ABB RobotStudio station: RAPID Project.rspag

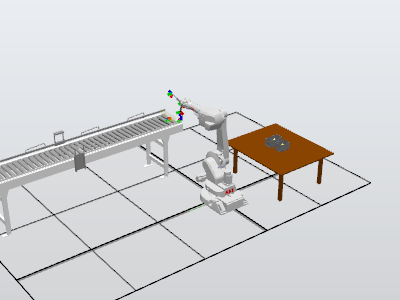
--- station ---
Station RAPID Project (saved by RobotStudio 23.4.10609.1)
Controller IRB1600_6_145
  mechanical unit ROB_1: IRB1600_6_145__03, 6 joints, base frame (0, 0, 0) mm
Layout (positions relative to the parent item):
  - IRB1600_6_145__03 [mechanism, from %ABB.RobotStudio.Models.IRB1600%\IRB1600_6_145_G_03.rslib] at (0, 0, 0) mm; joint values [0, 0, 0, 0, 0.5236, 0] (rad or m)
  - VacuumPenToolSC [smart component, from RAPID Project\VacuumPenToolSC.rslib] at (806.29, 0, 1154) mm, rotated rx 180 ry 60 rz 180 deg
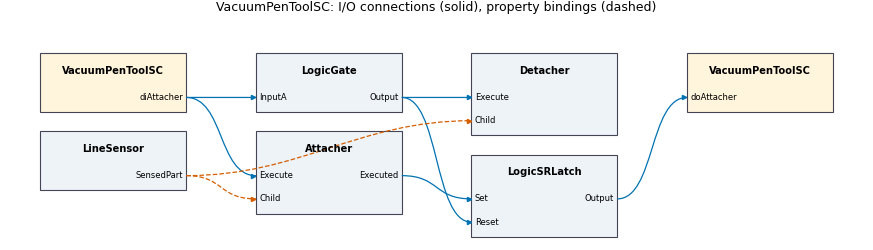
      connections:
        VacuumPenToolSC.diAttacher -> LogicGate.InputA
        LogicGate.Output -> Detacher.Execute
        Attacher.Executed -> LogicSRLatch.Set
        LogicSRLatch.Output -> VacuumPenToolSC.doAttacher
        VacuumPenToolSC.diAttacher -> Attacher.Execute
        LogicGate.Output -> LogicSRLatch.Reset
        LineSensor.SensedPart => Attacher.Child
        LineSensor.SensedPart => Detacher.Child
    - VacuumPenTool [mechanism, from RAPID Project\VacuumPenToolSC.rslib] at (0, 0, 0) mm
    - LineSensor [smart component, from Components\LineSensor.rslib]
        properties: Start=[0.107 -0.00037 0.127]; End=[0.114 0 0.134]; Radius=0.001; SensedPart=(none); SensedPoint=[0 0 0]; Length=0.00990640701768306; Tag=(none)
      - _sensorPart_ [part], size 8.4 x 2.4 x 8.4 mm
    - Attacher [smart component, from Components\Attacher.rslib]
        properties: Parent=VacuumPenTool; Flange=0; Child=(none); Mount=false; Offset=[0 0 0]; Orientation=[0 0 0]
    - Detacher [smart component, from Components\Detacher.rslib]
        properties: Child=(none); KeepPosition=true
    - LogicGate [smart component, from Components\LogicGate.rslib]
        properties: Operator=NOT; Delay=0
    - LogicSRLatch [smart component, from Components\LogicSRLatch.rslib]
  - mesa_marron [part] at (500, -500, 500) mm, rotated rx 90 ry 0 rz 180 deg, size 1200 x 500 x 1000 mm
  - box_big [part] at (1475.92, 2958.99, 0) mm, size 100 x 100 x 100 mm
  - box_small [part] at (1082.53, 3022.45, 0) mm, size 80 x 80 x 80 mm
  - Cardboard_container_bigSC [smart component]
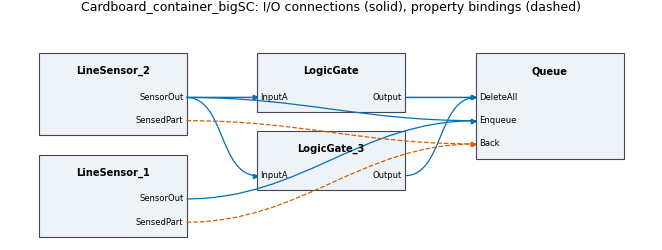
      connections:
        LineSensor_2.SensorOut -> LogicGate.InputA
        LogicGate.Output -> Queue.DeleteAll
        LineSensor_2.SensorOut -> LogicGate_2.InputA
        LogicGate_2.Output -> Queue.DeleteAll
        LineSensor_1.SensorOut -> Queue.Enqueue
        LineSensor_2.SensorOut -> Queue.Enqueue
        LineSensor_2.SensorOut -> LogicGate_3.InputA
        LogicGate_3.Output -> Queue.DeleteAll
        LineSensor_2.SensedPart => Queue.Back
        LineSensor_1.SensedPart => Queue.Back
    - UMS5_Cardboard_box_big_bottom [part] at (0, -1000, 521) mm, rotated rx 0 ry 0 rz -90 deg, size 220.2 x 110.8 x 110.2 mm
    - Queue [smart component, from Components\Queue.rslib]
        properties: Back=(none); Front=(none); Queue={6b8558fe-eb23-4042-ac4d-4b2e4693563e};{5ffcd9c3-88d3-497d-8378-cfc202dc5907};{29bb7ccf-0bc1-48a2-9f08-b9b634dbc6ca}; NumberOfObjects=1
    - LineSensor_1 [smart component, from Components\LineSensor.rslib]
        properties: Start=[0.05 -0.95 0.571]; End=[-0.05 -0.95 0.571]; Length=0.1; Radius=0; Tag=(none); SensedPart=(none); SensedPoint=[0.0499339485168457 -0.95 0.571]
      - _sensorPart_ [part], size 100 x 0 x 0 mm
    - LineSensor_2 [smart component, from Components\LineSensor.rslib]
        properties: Start=[0.05 -1.05 0.572]; End=[-0.05 -1.05 0.572]; Length=0.1; Radius=0; Tag=(none); SensedPart=(none); SensedPoint=[0 0 0]
      - _sensorPart_ [part], size 100 x 0 x 0 mm
    - LogicGate_3 [smart component, from Components\LogicGate.rslib]
        properties: Operator=NOP; Delay=4
  - Cardboard_container_smallSC [smart component]
      connections:
        LineSensor_3.SensorOut -> Queue_2.Enqueue
        LineSensor_4.SensorOut -> Queue_2.Enqueue
        LineSensor_4.SensorOut -> LogicGate_4.InputA
        LogicGate_4.Output -> Queue_2.DeleteAll
        LineSensor_3.SensedPart => Queue_2.Back
        LineSensor_4.SensedPart => Queue_2.Back
    - UMS5_Cardboard_box_small_bottom [part] at (-180, -1000, 521) mm, rotated rx 0 ry 0 rz -90 deg, size 180.2 x 110.8 x 110.2 mm
    - LineSensor_3 [smart component, from Components\LineSensor.rslib]
        properties: Start=[-0.23 -0.96 0.572]; End=[-0.13 -0.96 0.572]; Length=0.1; Radius=0; Tag=(none); SensedPart=(none); SensedPoint=[0 0 0]
      - _sensorPart_ [part], size 100 x 0 x 0 mm
    - LineSensor_4 [smart component, from Components\LineSensor.rslib]
        properties: Start=[-0.23 -1.04 0.572]; End=[-0.13 -1.04 0.572]; Length=0.1; Radius=0; Tag=(none); SensedPart=(none); SensedPoint=[0 0 0]
      - _sensorPart_ [part], size 100 x 0 x 0 mm
    - Queue_2 [smart component, from Components\Queue.rslib]
        properties: Back=(none); Front=(none); Queue=; NumberOfObjects=0
    - LogicGate_4 [smart component, from Components\LogicGate.rslib]
        properties: Operator=NOP; Delay=4
  - Conveyor [smart component] at (956.12, 2916.39, 0) mm, rotated rx 0 ry 0 rz -90 deg
      signals: DI start_or_resume, DO cube_ready, DO small_out, DO big_out
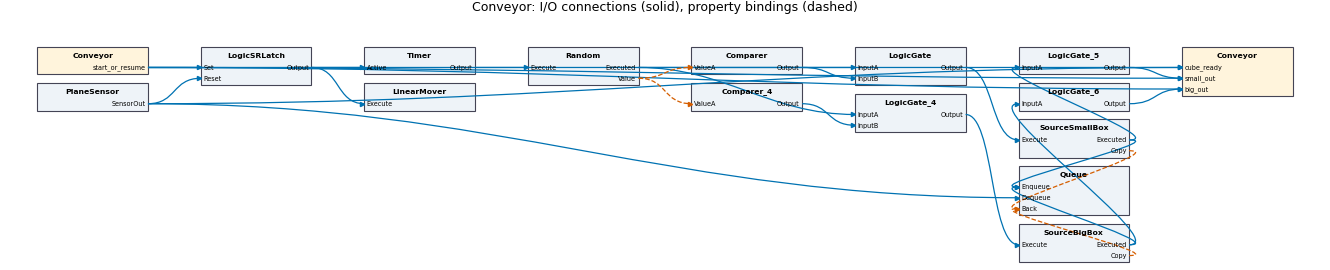
      connections:
        Timer.Output -> Random.Execute
        Random.Executed -> LogicGate.InputA
        Comparer.Output -> LogicGate.InputB
        Random.Executed -> LogicGate_4.InputA
        Comparer_4.Output -> LogicGate_4.InputB
        LogicGate.Output -> SourceSmallBox.Execute
        LogicGate_4.Output -> SourceBigBox.Execute
        SourceSmallBox.Executed -> Queue.Enqueue
        SourceBigBox.Executed -> Queue.Enqueue
        Conveyor.start_or_resume -> LogicSRLatch.Set
        PlaneSensor.SensorOut -> Queue.Dequeue
        PlaneSensor.SensorOut -> LogicSRLatch.Reset
        LogicSRLatch.Output -> Timer.Active
        LogicSRLatch.Output -> LinearMover.Execute
        PlaneSensor.SensorOut -> Conveyor.cube_ready
        SourceSmallBox.Executed -> LogicGate_5.InputA
        LogicGate_5.Output -> Conveyor.small_out
        SourceBigBox.Executed -> LogicGate_6.InputA
        LogicGate_6.Output -> Conveyor.big_out
        Conveyor.start_or_resume -> Conveyor.small_out
        Conveyor.start_or_resume -> Conveyor.big_out
        Conveyor.start_or_resume -> Conveyor.cube_ready
        Random.Value => Comparer.ValueA
        Random.Value => Comparer_4.ValueA
        SourceSmallBox.Copy => Queue.Back
        SourceBigBox.Copy => Queue.Back
    - SourceSmallBox [smart component, from Components\Source.rslib]
        properties: Source=box_small; Copy=(none); Parent=(none); Position=[1.118659 0.4 0.775]; Orientation=[0 0 0]; Transient=false; PhysicsBehavior=-1
    - SourceBigBox [smart component, from Components\Source.rslib]
        properties: Source=box_big; Copy=(none); Parent=(none); Position=[1.118659 0.4 0.775]; Orientation=[0 0 0]; Transient=false; PhysicsBehavior=-1
    - Random [smart component, from Components\Random.rslib]
        properties: Value=1.6316647863163; Min=0; Max=2
    - Comparer [smart component, from Components\Comparer.rslib]
        properties: ValueA=1.6316647863163; Operator=<=; ValueB=1
    - Timer [smart component, from Components\Timer.rslib]
        properties: StartTime=0; Interval=8; Repeat=true; CurrentTime=9.936
    - LogicGate [smart component, from Components\LogicGate.rslib]
        properties: Operator=AND; Delay=0
    - LogicGate_4 [smart component, from Components\LogicGate.rslib]
        properties: Operator=AND; Delay=0
    - Comparer_4 [smart component, from Components\Comparer.rslib]
        properties: ValueA=1.6316647863163; Operator=>; ValueB=1
    - Queue [smart component, from Components\Queue.rslib]
        properties: Back=(none); Front=(none); Queue={1131f909-5d82-4e84-bc9f-120231f9d299};{405f4df7-07e7-4b74-a1a1-a810a0d8cfa6};{743c33c0-6a87-4aec-9895-952089b91bbd};{216fa1ae-755b-4613-beaf-a983367b2fa7};{bf1b47c8-f294-4567-aa47-23f27967580f};{64bd0bdc-0a47-47ab-a397-a74a684aee1e};{437488d7-8282-475b-b486-389db32fdaa2};{671afbe1-b4fc-4869-acfd-eeadac196f1e};{a4dc94ab-7dff-4b2f-b405-15f84814c83e};{c4b58b1b-6de3-44d8-9367-5c715bdef502};{dda5cb65-1224-402a-bab3-4bfeb52fa140};{8990a0b7-37dc-4b49-b0cf-ca37f5f81eb5};{063f5e72-8178-40bf-9af7-13761aa78818};{318b9655-dbdc-41bc-a948-0739e52a5f4e};{94459ab9-d214-4441-90b7-aab42f321ec1};{846e7d94-1788-41a0-bce8-b7df51ff760f};{16d7a3a2-3dec-478f-b63b-07f1d7cc03de};{580626d5-5194-432f-9920-3f632f566f7d};{09cd6ac9-05a0-4cd8-820b-7021498e93a7};{8b0e4d5d-dbbf-4476-8b58-1e0bb391d2bd};{72ea86c5-dea0-4016-afa7-4ec3a2f95cb2};{db5153cf-1ef7-4663-8b40-1eb38a32e43d};{b4adc6ae-5d32-4435-8d0a-f83dcca57720};{47c401ac-b51c-4c6d-9a18-a43309c02b6f};{a14179fa-a620-42e3-b84a-d28d3825529b};{75bd4498-393a-48f7-a61b-542cce98fff7};{a0be46a5-9209-4291-b80b-03db147a5a1d};{62579eb4-f161-4662-b633-27fb85a22197};{8ab14ceb-fd47-4ba4-a6bd-d5a5c6825a1f};{2bf3086a-31c6-43ba-81ac-83cd6e2c523b};{178fb3f7-54e1-49b5-b854-21d9b4cccd97};{60c9e6ba-6b64-485d-ac32-6a969e7af7d0};{e716be99-0149-4cae-beca-e0cc469dbdf1};{1ed01c8b-55dc-4a17-92b3-7dcc16efebbf};{0c751f24-0e05-4f2d-a7e6-2b57fe9a78f8};{6bdb1028-fc23-4fb2-bfed-e8dd47b3d521};{8032889f-a66e-44c4-87e0-11a35d7802f5};{e82d9fc5-fcd6-414b-8dbe-c18ec15ec5e2};{ef39c74a-18b4-4780-ad05-efc2b3f11d14};{1f129472-405d-47d1-9b42-e2634ee9a6ca};{d99a7689-406e-4b3a-acdb-2f92a8b49675};{762a0486-21c4-4276-88c3-fe9305565678};{518b26eb-ac13-4676-a60e-00d758036b53};{f3293468-b94e-4e49-8e4d-c35ec2676aa0};{968cdc0a-45a6-417b-877a-2dca0b94f2dc};{2307791a-20a1-4e9f-a50a-49ddd01e3173};{669990e8-965e-434c-afe6-05f7427a6bd7};{f660ccc2-823d-4eb9-99d0-62b29f80a269};{2c39a5b9-3e01-400d-97c7-1b6ddbd0b428};{3e5914c8-bfd0-4d5d-b879-bcb13d1fe68a};{9d29d2dc-6e76-4714-8490-c2a022750207};{84804570-8629-4e0c-8c93-96a2edbbd09e};{063ecb17-a126-4a64-bc2e-c236ff422495};{d5eda05f-c4af-43ea-a80f-10962ebe72cb};{dba58393-be63-4a9b-a3f9-785f42c24db6};{6b8558fe-eb23-4042-ac4d-4b2e4693563e};{40838503-966e-44b9-9226-e66a6092ff01};{226e4f7c-7e9b-486a-b901-bcc49bf84f10};{0beb15ee-4784-4d3f-af16-8f4a4751a885};{11c0db58-aac9-483f-9d7b-0be503b7f118};{21889f9e-5f6e-4675-a0f6-b8030afa24f2};{2ec464fe-71d2-4c92-b6a8-21ae5a9722c9};{0079b514-c3c4-4a73-84ee-0bac4bec86eb};{37d905e1-bf83-4712-a54d-8ee25133736b};{32e9c903-d330-495a-9fd7-b7ae14ea847b};{80be3bce-579e-4408-a68f-69d701d026d4};{463f11c4-1cdc-43ce-ab84-5d6c25b7273d};{ad7a2bf7-7240-4966-9c51-4ffcbb69f75a};{5ffcd9c3-88d3-497d-8378-cfc202dc5907};{9d4476dd-9eba-40a7-b40c-6b531b19a73b};{e032135e-4a59-4f03-926c-afd51edca3d8};{5d2df8e7-df73-4e08-bee6-4ebbf4db4217};{29bb7ccf-0bc1-48a2-9f08-b9b634dbc6ca}; NumberOfObjects=0
    - LinearMover [smart component, from Components\LinearMover.rslib]
        properties: Object=Queue; Direction=[0 -0.5 0]; Speed=0.06; Reference=Global; ReferenceObject=(none)
    - PlaneSensor [smart component, from Components\PlaneSensor.rslib]
        properties: Origin=[2.910135 0.39 0.78]; Axis1=[0 -0.38 0]; Axis2=[0 0 0.1]; Tag=(none); SensedPart=(none)
      - _sensorPart_ [part], size 0 x 380 x 100 mm
    - LogicSRLatch [smart component, from Components\LogicSRLatch.rslib]
    - 400_guide [part], size 3033 x 590 x 945 mm
    - LogicGate_5 [smart component, from Components\LogicGate.rslib]
        properties: Operator=NOT; Delay=0
    - LogicGate_6 [smart component, from Components\LogicGate.rslib]
        properties: Operator=NOT; Delay=0
  - EMERGENCY_STOP [smart component]
      signals: DO EMERGENCY_STOP
Attachment: VacuumPenToolSC is attached to IRB1600_6_145__03 / Link6
Station logic (signal -> signal, property => property):
  IRB1600_6_145.vacuum -> VacuumPenToolSC.diAttacher
  Conveyor.small_out -> IRB1600_6_145.small
  Conveyor.big_out -> IRB1600_6_145.big
  Conveyor.cube_ready -> IRB1600_6_145.cube_ready
  IRB1600_6_145.Resume -> Conveyor.start_or_resume
  EMERGENCY_STOP.EMERGENCY_STOP -> IRB1600_6_145.em_stop
Targets, tools, work objects and paths stored in the station and not in the controller backup, written as RAPID:
! task T_ROB1
MODULE Module1
  CONST robtarget pplace:=[[0,0,0],[1,0,0,0],[0,0,0,0],[9E+09,9E+09,9E+09,9E+09,9E+09,9E+09]];
ENDMODULE


--- Controller Data/IRB1600_6_145/RAPID/TASK1/PROGMOD/Module1.mod ---
MODULE Module1
    PERS tooldata VacuumTool:=[TRUE,[[106.338,-0.37,126.015],[0.923879533,0,0.382683432,0]],[1,[0,0,1],[1,0,0,0],0,0,0]];
    PERS tooldata PenTool:=[TRUE,[[-174.289,-0.18,194.277],[0.923879533,0,-0.382683432,0]],[1,[0,0,1],[1,0,0,0],0,0,0]];

    VAR intnum emergency;
    VAR intnum em_continue;

    VAR num number_of_boxes{2}:=[0,0];

    CONST num off_flyby:=-150;
    CONST num off_approach:=-75;

    CONST speeddata v_safe:=v300;
    CONST speeddata v_approach:=v100;
    CONST speeddata v_draw:=v50;
    CONST speeddata v_place:=v50;

    CONST robtarget home1:=[[1061.684968927,-0.18,1207.800197059],[0.793353336,0,0.608761435,0],[-1,0,-1,0],[9E+09,9E+09,9E+09,9E+09,9E+09,9E+09]];
    VAR robtarget pwobj1_draw:=[[0,0,0],[0,0,0,1],[0,0,0,0],[9E+09,9E+09,9E+09,9E+09,9E+09,9E+09]];
    CONST robtarget pwobj2_place:=[[0,0,0],[0,0,1,0],[-3,0,0,0],[9E+09,9E+09,9E+09,9E+09,9E+09,9E+09]];

    PERS wobjdata wobj_conv:=[FALSE,TRUE,"",[[956.122,-83.614,800],[1,0,0,0]],[[162.54,88.96,-25.00],[0.707106781,0,0.707106781,0]]];
    PERS wobjdata wobj_table:=[FALSE,TRUE,"",[[500.00,-500.00,520.00],[0,0,0,1]],[[600,500,1],[0.7071,0,0,0.7071]]];

    PROC main()
        !Connect interrupts to TRAP functions
        CONNECT emergency WITH Emergency_Stop;
        CONNECT em_continue WITH Emergency_Continue;

        !Order interupts from digital input signals

        !Signal for an emergency stop
        ISignalDI em_stop,1,emergency;

        !Signal for continuing after an emergency stop
        ISignalDI em_stop,0,em_continue;

        !Reset every signal from the conveyor before starting
        PulseDO Resume;
        WaitTime 1;

        !Iterative process of drawing and palletizing pill boxes
        FOR i FROM 0 TO 10 DO

            !Resetting the number of boxes from the cardboard containers (maximum is 2)
            Reset_number number_of_boxes;

            !Waiting until the box is in position on the conveyor
            WaitUntil TestDI(cube_ready);

            !Checking size of the box
            IF DInput(big)=1 THEN
                Big_box;
            ELSEIF DInput(small)=1 THEN
                Small_box;
            ENDIF
        ENDFOR

    ENDPROC

    !Routine for the big box
    PROC Big_box()

        !Making sure the vaccum is off
        SetDO vacuum, 0;
        Draw 100;
        Pick_place 100, pwobj1_draw, number_of_boxes{1};

        !Incrementing the number of boxes from the cardboard containers
        number_of_boxes{1} := number_of_boxes{1} + 1;
    ENDPROC

    !Routine for the small box
    PROC Small_box()

        !Making sure the vaccum is off
        SetDO vacuum, 0;

        Draw -80;
        Pick_place -80, pwobj1_draw, number_of_boxes{2};

        !Incrementing the number of boxes from the cardboard containers
        number_of_boxes{2} := number_of_boxes{2} + 1;
    ENDPROC

    PROC Draw(num box_length)
        MoveJ home1,v1000,z100,PenTool\WObj:=wobj0;

        !Approach point
        MoveJ Offs(pwobj1_draw,-Abs(box_length/2),Abs(box_length/8), off_flyby),v_safe,z50,PenTool\WObj:=wobj_conv;
        MoveL Offs(pwobj1_draw,-Abs(box_length/2),Abs(box_length/8), off_approach),v_approach,z10,PenTool\WObj:=wobj_conv;

        !Move to draw point
        MoveL Offs(pwobj1_draw,-Abs(box_length/2),Abs(box_length/8), 0), v_draw,fine,PenTool\WObj:=wobj_conv;
        MoveC Offs(pwobj1_draw,-Abs(box_length/2)+box_length/8,Abs(box_length/2),0), Offs(pwobj1_draw,-Abs(box_length/2),Abs(box_length-box_length/8),0), v_draw, fine, PenTool\WObj:=wobj_conv;
        MoveL Offs(pwobj1_draw,-Abs(box_length/2),Abs(box_length/8), 0), v_draw,fine,PenTool\WObj:=wobj_conv;

        MoveL Offs(pwobj1_draw,-Abs(box_length/2),Abs(box_length/8), off_approach),v_approach,z10,PenTool\WObj:=wobj_conv;
        MoveJ Offs(pwobj1_draw,-Abs(box_length/2),Abs(box_length/8), off_flyby),v_safe,z50,PenTool\WObj:=wobj_conv;

        MoveJ home1,v1000,z100,PenTool\WObj:=wobj0;
    ENDPROC

    PROC Pick_place(num box_length, robtarget point, num number_boxes)

        !Changing orentation for "pwobj1_draw" to suit the operations of the vacuum
        point.rot:=[0.7071,0, 0.7071,0];

        MoveJ home1,v1000,z100,PenTool\WObj:=wobj0;

        !Approach point
        MoveJ Offs(point,-Abs(box_length)+off_approach,Abs(box_length)/2,Abs(box_length)/2),v_safe,z10,VacuumTool\WObj:=wobj_conv;

        !Move to pick point
        MoveL Offs(point,-Abs(box_length)-3,Abs(box_length)/2,Abs(box_length)/2),v_approach,fine,VacuumTool\WObj:=wobj_conv;
        Pick;
        MoveL Offs(point,-Abs(box_length)+off_approach,Abs(box_length)/2,Abs(box_length)/2),v_safe,z10,VacuumTool\WObj:=wobj_conv;

        !Generating the next block while palletizing
        PulseDO Resume;

        MoveJ Offs(pwobj2_place,-Abs(box_length/2)+number_boxes*(Abs(box_length) + 2),box_length,300), v1000,z10,VacuumTool\WObj:=wobj_table;
        MoveJ Offs(pwobj2_place,-Abs(box_length/2)+number_boxes*(Abs(box_length) + 2),box_length,-off_flyby), v_approach,fine,VacuumTool\WObj:=wobj_table;
        MoveL Offs(pwobj2_place,-Abs(box_length/2)+number_boxes*(Abs(box_length) + 2),box_length,Abs(box_length)+2), v_place,fine,VacuumTool\WObj:=wobj_table;
        Place;

        MoveJ Offs(pwobj2_place,-Abs(box_length/2)+number_boxes*(Abs(box_length) + 2),box_length,-off_flyby), v_approach,fine,VacuumTool\WObj:=wobj_table;

        MoveJ home1,v1000,z100,PenTool\WObj:=wobj0;
    ENDPROC

    !Picking routine
    PROC Pick()
        SetDO vacuum, 1;
        WaitTime 1;
    ENDPROC

    !Placing routine
    PROC Place()
        SetDO vacuum, 0;
        WaitTime 1;
    ENDPROC

    !Resetting the number of the pill boxes from the carboard containers
    PROC Reset_number(VAR num number_boxes{*})
        IF number_boxes{1}=2 THEN
            number_boxes{1}:=0;
        ENDIF
        IF number_boxes{2}=2 THEN
            number_boxes{2}:=0;
        ENDIF
    ENDPROC

    TRAP Emergency_Stop
        !Stops the movement of the robot
        StopMove;
        RETURN;
    ENDTRAP

    TRAP Emergency_Continue
        !Resumes the trajectory of the robot
        StartMove;
        RETURN;
    ENDTRAP

ENDMODULE

--- Controller Data/IRB1600_6_145/SYSPAR/EIO.cfg ---
EIO:CFG_1.0:6:1::
#
EIO_SIGNAL:

      -Name "vacuum" -SignalType "DO"

      -Name "small" -SignalType "DI"

      -Name "big" -SignalType "DI"

      -Name "cube_ready" -SignalType "DI"

      -Name "Resume" -SignalType "DO"

      -Name "em_stop" -SignalType "DI"
